// TIA Portal V17 export
// export: Created 2023-02-13T11:16:45.5062183Z, ExportSetting WithDefaults, DisplayName Totally Integrated Automation Portal, DisplayVersion V17, DisplayName TIA Portal Openness, DisplayVersion V17, DisplayName TIA Portal Teamcenter Gateway, DisplayVersion V17, DisplayName TIA Portal Version Control Interface, DisplayVersion V17, DisplayName SINAMICS Startdrive Advanced, DisplayVersion V17, DisplayName SINAMICS Startdrive G130, G150, S120, S150, SINAMICS MV, S210, DisplayVersion V17, DisplayName SINAMICS Startdrive G110M, G120, G120C, G120D, G120P, G115D, DisplayVersion V17, DisplayName STEP 7 Professional, DisplayVersion V17, DisplayName STEP 7 Safety, DisplayVersion V17, DisplayName WinCC Professional, DisplayVersion V17
FUNCTION "Pulse" : Void   // FC10, LAD
{ S7_Optimized_Access := 'TRUE' }
VERSION : 0.1
// stored: AutoNumber true, IsIECCheckEnabled false, SetENOAutomatically false, UDAEnableTagReadback false
   VAR_TEMP   // added for the SCL form of the ladder/FBD networks
      _w1 : Bool;
      _s5time1 : S5Time;
      _w2 : Bool;
      _s5time2 : S5Time;
   END_VAR
BEGIN

REGION Network 1: Timer 5s/ 1M
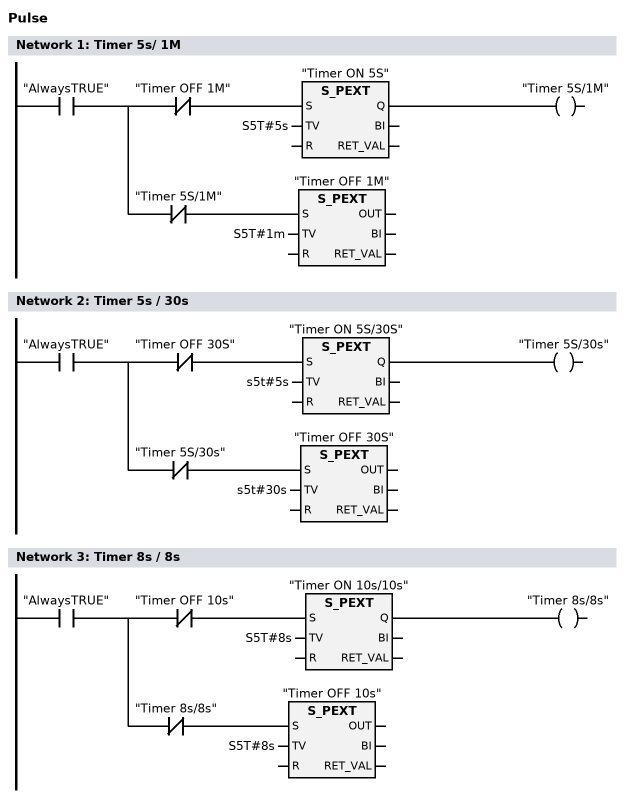
   RUNG wire#powerrail
      Contact( "AlwaysTRUE" )
      wire#w1
      I_Contact( "Timer OFF 1M" )
      S_PEXT(T_NO := "Timer ON 5S", TV := S5T#5s, R :=, BI =>, RET_VAL =>)
      Coil( "Timer 5S/1M" )
   END_RUNG
   RUNG wire#w1
      I_Contact( "Timer 5S/1M" )
      S_PEXT(T_NO := "Timer OFF 1M", TV := S5T#1m, R :=, BI =>, RET_VAL =>)
   END_RUNG
   // the same network as SCL:
   #_w2 := "AlwaysTRUE";
   #_s5time1 := S_PEXT(T_NO := "Timer ON 5S", S := "AlwaysTRUE" AND NOT "Timer OFF 1M", TV := S5T#5s, Q => #_w1);
   "Timer 5S/1M" := #_w1;
   #_s5time2 := S_PEXT(T_NO := "Timer OFF 1M", S := #_w2 AND NOT "Timer 5S/1M", TV := S5T#1m);
END_REGION

REGION Network 2: Timer 5s / 30s
   RUNG wire#powerrail
      Contact( "AlwaysTRUE" )
      wire#w1
      I_Contact( "Timer OFF 30S" )
      S_PEXT(T_NO := "Timer ON 5S/30S", TV := s5t#5s, R :=, BI =>, RET_VAL =>)
      Coil( "Timer 5S/30s" )
   END_RUNG
   RUNG wire#w1
      I_Contact( "Timer 5S/30s" )
      S_PEXT(T_NO := "Timer OFF 30S", TV := s5t#30s, R :=, BI =>, RET_VAL =>)
   END_RUNG
   // the same network as SCL:
   #_w2 := "AlwaysTRUE";
   #_s5time1 := S_PEXT(T_NO := "Timer ON 5S/30S",
                       S := "AlwaysTRUE" AND NOT "Timer OFF 30S",
                       TV := s5t#5s,
                       Q => #_w1);
   "Timer 5S/30s" := #_w1;
   #_s5time2 := S_PEXT(T_NO := "Timer OFF 30S", S := #_w2 AND NOT "Timer 5S/30s", TV := s5t#30s);
END_REGION

REGION Network 3: Timer 8s / 8s
   RUNG wire#powerrail
      Contact( "AlwaysTRUE" )
      wire#w1
      I_Contact( "Timer OFF 10s" )
      S_PEXT(T_NO := "Timer ON 10s/10s", TV := S5T#8s, R :=, BI =>, RET_VAL =>)
      Coil( "Timer 8s/8s" )
   END_RUNG
   RUNG wire#w1
      I_Contact( "Timer 8s/8s" )
      S_PEXT(T_NO := "Timer OFF 10s", TV := S5T#8s, R :=, BI =>, RET_VAL =>)
   END_RUNG
   // the same network as SCL:
   #_w2 := "AlwaysTRUE";
   #_s5time1 := S_PEXT(T_NO := "Timer ON 10s/10s",
                       S := "AlwaysTRUE" AND NOT "Timer OFF 10s",
                       TV := S5T#8s,
                       Q => #_w1);
   "Timer 8s/8s" := #_w1;
   #_s5time2 := S_PEXT(T_NO := "Timer OFF 10s", S := #_w2 AND NOT "Timer 8s/8s", TV := S5T#8s);
END_REGION
END_FUNCTION
